(* IEC 61131-3 sources: SRCI/RobotLibrary/Library/POUs/_internal/LogFBs, 1 file *)

(* ---- AxesGroupMessageLogFB.st ---- *)
FUNCTION_BLOCK AxesGroupMessageLogFB IMPLEMENTS IMessageLogger
// -------------------------------------------------------------------------
//  SRCI Robot Library
// -------------------------------------------------------------------------
//
//  Object:      AxesGroupMessageLogFB
//  Author:      Thorsten Brach
//  Date:        2025-01-05
//
//  Description:
//
//
//  Copyright:
//    (C) 2025 Thorsten Brach. All rights reserved
//             Licensed under the LGPL-3.0 license.
//
//  Disclaimer:
//    This project is provided without any guarantee and can be used for
//    private and commercial purposes. Any use is at the user’s
//    own risk and responsibility.
//
// -------------------------------------------------------------------------
VAR_INPUT
  /// Logging level
  LogLevel         : LogLevel;
  /// Interface to an external logger
  ExternalLogger   : IMessageLogger;
END_VAR

VAR_OUTPUT
  /// Amount of system log entries
  SystemLogEntries : UINT := 0;
  /// Amount of message log entries
  MessagesEntries  : UINT := 0;
  /// System log
  SystemLogs       : ARRAY[0..RobotLibraryParameter.SYSTEM_LOG_MAX ] OF STRING(RobotLibraryParameter.MESSAGE_TEXT_LEN);
  /// Message Log
  Messages         : ARRAY[0..RobotLibraryParameter.MESSAGE_LOG_MAX] OF AlarmMessage;
END_VAR

END_FUNCTION_BLOCK

METHOD PUBLIC AddMessageLog
VAR_INPUT
  MessageLog : AlarmMessage;
END_VAR

VAR
  /// internal index
 _idx            : DINT;
  /// internal index to delete
 _idxFound       : DINT;
  /// lowest Severity
 _lowestSeverity : Severity := Severity.FATAL_ERROR;
  /// temporary buffer ( must be one element less than the message log !!! )
 _tmpBuffer      : ARRAY[0..RobotLibraryParameter.MESSAGE_LOG_MAX -1] OF AlarmMessage;
END_VAR

  // Check entry must be added ?
  IF (( LogLevel  <= MessageLog.Severity     ) AND
      ( LogLevel  >  LogLevelEnum.DEACTIVATE ))
  THEN
    // Check message buffer is full ?
    IF ( MessagesEntries >= RobotLibraryParameter.MESSAGE_LOG_MAX )
    THEN
      // find lowest Severity
      FOR _idx := 1 TO RobotLibraryParameter.MESSAGE_LOG_MAX
      DO
        // check entry has a lower severity ?
       _lowestSeverity := MIN( Messages[_idx].Severity, _lowestSeverity );
  		END_FOR

      // search for the oldes message with a lower Severity
      FOR _idx := RobotLibraryParameter.MESSAGE_LOG_MAX TO 1 BY -1
      DO
        // message found ?
        IF (( Messages[_idx].Severity <   MessageLog.Severity ) AND
            ( Messages[_idx].Severity <= _lowestSeverity      ))
        THEN
          // save index to delete
         _idxFound := _idx;
          EXIT;
  			END_IF
  		END_FOR

      // check message must be deleted ?
      IF ( _idxFound > 0 )
      THEN
        // shift all messages starting from the found index one position forwards
        FOR _idx := _idxFound TO RobotLibraryParameter.MESSAGE_LOG_MAX -1
        DO
          Messages[_idx] := Messages[_idx +1];
  			END_FOR
  		END_IF
    END_IF

    // shift all messages one position backwards
    // shift messages log entries
    SysDepMemCpy( pDest := ADR(_tmpBuffer[0]), pSrc := ADR(  Messages[0]), DataLen := SIZEOF(_tmpBuffer));
    SysDepMemCpy( pDest := ADR(  Messages[1]), pSrc := ADR(_tmpBuffer[0]), DataLen := SIZEOF(_tmpBuffer));

    // Add new message
    Messages[0].Timestamp   := MessageLog.Timestamp;
    Messages[0].MessageType := MessageLog.MessageType;
    Messages[0].Severity    := MessageLog.Severity;
    Messages[0].MessageText := MessageLog.MessageText;
    Messages[0].MessageCode := MessageLog.MessageCode;

    // inc message counter
    MessagesEntries := DINT_TO_UINT(LIMIT(0, MessagesEntries + 1, RobotLibraryParameter.MESSAGE_LOG_MAX));
  END_IF

END_METHOD

METHOD Public AddMessageLogByParameter
VAR_INPUT
  /// Timestamp
  Timestamp   : SystemTime;
  /// Type of message according to Table 5-46:
  MessageType : MessageType;
  /// Severity of message according to Table 5-47: Debug, Info, Warning, Error, Fatal error
  Severity    : Severity;
  /// Code of messages
  MessageCode : DWORD;
  /// Static text of message
  MessageText : STRING(RobotLibraryParameter.MESSAGE_TEXT_LEN);
END_VAR

VAR
  /// temporary message
 _message : AlarmMessage;
END_VAR

  _message.Timestamp   := Timestamp;
  _message.MessageType := MessageType;
  _message.MessageCode := MessageCode;
  _message.MessageText := MessageText;
  _message.Severity    := Severity;

  // Add message to message buffer
  AddMessageLog(_message);

END_METHOD

METHOD PUBLIC AddSystemLog
VAR_INPUT
  /// system log message
  SystemLog : STRING(255);
END_VAR
VAR
  /// internal index
 _idx       : DINT;
  /// internal log message
 _message   : AlarmMessage;
  /// temporary buffer ( must be one element less than the system log !!! )
 _tmpBuffer : ARRAY[0..RobotLibraryParameter.SYSTEM_LOG_MAX -1] OF STRING(RobotLibraryParameter.MESSAGE_TEXT_LEN);
END_VAR

  // shift system log entries
  SysDepMemCpy( pDest := ADR(_tmpBuffer[0]), pSrc := ADR(SystemLogs[0]), DataLen := SIZEOF(_tmpBuffer));
  SysDepMemCpy( pDest := ADR(SystemLogs[1]), pSrc := ADR(_tmpBuffer[0]), DataLen := SIZEOF(_tmpBuffer));

  // Delete CR from system log message
  SystemLog := StrReplace(SystemLog, '$R', '');
  // Delete LF from system log message
  SystemLog := StrReplace(SystemLog, '$N', '');

  // Add System log to buffer
  SystemLogs[0] := SystemLog;

  // inc SystemLog counter
  SystemLogEntries := DINT_TO_UINT(LIMIT(0, SystemLogEntries + 1, RobotLibraryParameter.SYSTEM_LOG_MAX));

END_METHOD

METHOD CheckMessageCodePresent : BOOL
VAR_INPUT
  /// Code of messages
  MessageCode : DWORD;
END_VAR

VAR
  /// internal index for loops
 _idx : DINT;
END_VAR

  FOR _idx := 0 TO RobotLibraryParameter.MESSAGE_LOG_MAX
  DO
    IF (Messages[_idx].MessageCode = MessageCode)
    THEN
      CheckMessageCodePresent := TRUE;
      RETURN;
  	END_IF
  END_FOR

END_METHOD

METHOD PUBLIC DeleteMessages
VAR_INPUT
END_VAR

  // reset messages
  SysDepMemSet(ADR(Messages), 0, SIZEOF(Messages));
  // reset message counter
  MessagesEntries := 0;

END_METHOD

METHOD DeleteSystemLogs
VAR_INPUT
END_VAR

  // reset SystemLogs
  SysDepMemSet(ADR(SystemLogs), 0, SIZEOF(SystemLogs));
  // reset SystemLogs counter
  SystemLogEntries := 0;

END_METHOD
